// TIA Portal V17 export
// export: Created 2025-03-10T13:11:50.4849452Z, ExportSetting WithDefaults, DisplayName Totally Integrated Automation Portal, DisplayVersion V17 Update 8, DisplayName TIA Portal Openness, DisplayVersion V17 Update 8, DisplayName TIA Portal Version Control Interface, DisplayVersion V17, DisplayName SINAMICS Startdrive Advanced, DisplayVersion V17 SP2, DisplayName SINAMICS Startdrive G110M, G120, G120C, G120D, G120P, G115D, DisplayVersion V17 SP2, DisplayName SINAMICS Startdrive G130, G150, S120, S150, SINAMICS MV, S210, DisplayVersion V17 SP2, DisplayName STEP 7 Professional, DisplayVersion V17 Update 8, DisplayName SINUMERIK ONE STEP 7 Toolbox, DisplayVersion V17 Update 12, DisplayName SINUMERIK 840D sl STEP 7 Toolbox, DisplayVersion V17 Update 12, DisplayName STEP 7 Safety, DisplayVersion V17 Update 6, DisplayName WinCC Advanced, DisplayVersion V17 Update 8
VAR_GLOBAL   // PLC tag table "TAGS_IO_PROFINET_CLADDING"
   "/////_POWER_METER_/////" AT %M7000.0 : Bool;   // ///// POWER METER /////
   POWER_METER_TOTAL_APPARENT_FACTOR AT %MD7058 : Real;   // POWER METER TOTAL APPARENT FACTOR
   POWDER_METER_MAX_TOTAL_APPARENT_POWER AT %ID3560 : Real;   // POWDER METER MAX TOTAL APPARENT POWER
   POWER_FACTOR_L3 AT %ID3524 : Real;   // POWER FACTOR L3
   POWER_METER_ACTIVE_POWER_L3 AT %MD7046 : Real;   // POWER METER ACTIVE POWER L3
   POWER_METER_TOTAL_APPARENT_POWER AT %ID3532 : Real;   // POWER METEER TOTAL APPARENT POWER
   POWER_METER_ACTIVE_ENERGY_IMPORT_TARIFF_F AT %ID3536 : Real;   // POWER METER ACTIVE ENERGY IMPORT TARIFF (F)
   POWER_FACTOR_L1 AT %ID3516 : Real;   // POWER FACTOR L1
   POWER_METER_TOTAL_REACTIVE_POWER AT %ID3512 : Real;   // POWER METER TOTAL REACTIVE POWER
   POWER_METER_CURRENT_L3 AT %ID3556 : Real;   // POWER METER CURRENT L3
   POWER_METER_ACTIVE_ENERGY_IMPORT AT %MD7050 : Real;   // POWER METER ACTIVE ENERGY IMPORT TARRIF
   POWDER_METER_UNIVERSAL_COUNTER_1 AT %ID3544 : Real;   // POWDER METER UNIVERSAL COUNTER 1
   POWER_METER_ACTIVE_POWER_L1 AT %MD7038 : Real;   // POWER METER ACTIVE POWER L1
   POWER_METER_ACTIVE_POWER_L2 AT %MD7042 : Real;   // POWER METER ACTIVE POWER L2
   POWER_METER_ACTIVE_ENERGY_EXPORT_TARIFF_F AT %ID3540 : Real;   // POWER METER ACTIVE ENERGY EXPORT TARIFF (F)
   POWER_METER_TOTAL_ACTIVE_POWER AT %ID3528 : Real;   // POWER METER TOTAL ACTIVE POWER
   POWER_METER_CURRENT_L2 AT %ID3552 : Real;   // POWER METER CURRENT L2
   POWER_METER_CURRENT_L1 AT %ID3548 : Real;   // POWER METER CURRENT L1
   POWER_FACTOR_L2 AT %ID3520 : Real;   // POWER FACTOR L2
   POWER_METER_VOLTAGE_L2_L3 AT %ID3576 : Real;   // POWER METER VOLTAGE L2-L3
   POWER_METER_VOLTAGE_L2_N AT %ID3588 : Real;   // POWER METER VOLTAGE L2 N
   POWER_METER_VOLTAGE_L3_N AT %ID3592 : Real;   // POWER METER VOLTAGE L3 N
   POWER_METER_VOLTAGE_L1_N AT %ID3584 : Real;   // POWER METER VOLTAGE L1 N
   POWER_METER_LINE_FRECUENCY AT %ID3568 : Real;   // POWER METER LINE FRECUENCY
   POWER_METER_VOLTAGE_L3_L1 AT %ID3580 : Real;   // POWER METER VOLTAGE L3-L1
   POWER_METER_VOLTAGE_L1_L2 AT %ID3572 : Real;   // POWER METER VOLTAGE L1-L2
   POWER_METER_TOTAL_POWER_FACTOR AT %ID3564 : Real;   // POWER METER TOTAL POWER FACTOR
END_VAR
